		INDICATOR_FWE_BRG := FALSE;
		INDICATOR_FWE_MCR := FALSE;
		INDICATOR_FWE_LC := FALSE;
	(*current status is STANDBY*)
	ELSIF   AUX_EOT_STATUS = 1
	THEN
		(*All the “STAND BY” indicators should keep stable light*)
		INDICATOR_STANDBY_BRG := TRUE;
		INDICATOR_STANDBY_MCR := TRUE;
		INDICATOR_STANDBY_LC := TRUE;
		(*other indicators should keep light off*)
		INDICATOR_ATSEA_BRG := FALSE;
		INDICATOR_ATSEA_MCR := FALSE;
		INDICATOR_ATSEA_LC := FALSE;
		INDICATOR_FWE_BRG := FALSE;
		INDICATOR_FWE_MCR := FALSE;
		INDICATOR_FWE_LC := FALSE;
	(*current status is ATSEA*)
	ELSIF  AUX_EOT_STATUS = 2
	THEN
		(*All the “AT SEA” indicators should keep stable light*)
		INDICATOR_ATSEA_BRG := TRUE;
		INDICATOR_ATSEA_MCR := TRUE;
		INDICATOR_ATSEA_LC := TRUE;
		(*other indicators should keep light off*)
		INDICATOR_STANDBY_BRG := FALSE;
		INDICATOR_STANDBY_MCR := FALSE;
		INDICATOR_STANDBY_LC := FALSE;
		INDICATOR_FWE_BRG := FALSE;
		INDICATOR_FWE_MCR := FALSE;
		INDICATOR_FWE_LC := FALSE;
	(*current status is F.W.E*)
	ELSIF	AUX_EOT_STATUS = 3
	THEN
		(*All the 'FWE” indicators should keep stable light*)
		INDICATOR_FWE_BRG := TRUE;
		INDICATOR_FWE_MCR := TRUE;
		INDICATOR_FWE_LC := TRUE;
		(*other indicators should keep light off*)
		INDICATOR_STANDBY_BRG := FALSE;
		INDICATOR_STANDBY_MCR := FALSE;
		INDICATOR_STANDBY_LC := FALSE;
		INDICATOR_ATSEA_BRG := FALSE;
		INDICATOR_ATSEA_MCR := FALSE;
		INDICATOR_ATSEA_LC := FALSE;
	END_IF
END_IF


CASE AUX_EOT_STATUS OF
	(*none status*)
	0:	H_AT_SEA := FALSE;	(*PROEOT0003*)
		H_STAND_BY := FALSE;	(*PROEOT0004*)
		H_FINSHED_WITH_ENGINE := FALSE;	(*PROEOT0005*)
	(*STAND BY*)
	1:	H_AT_SEA := FALSE;
		H_STAND_BY := TRUE;
		H_FINSHED_WITH_ENGINE := FALSE;
	(*AT SEA*)
	2:	H_AT_SEA := TRUE;
		H_STAND_BY := FALSE;
		H_FINSHED_WITH_ENGINE := FALSE;
	(*FWE*)
	3:	H_AT_SEA := FALSE;
		H_STAND_BY := FALSE;
		H_FINSHED_WITH_ENGINE := TRUE;
END_CASE;
END_FUNCTION_BLOCK

(* POU MISMATCH_ALARM, ST *)
(*4.1.7.1.4*)
FUNCTION_BLOCK MISMATCH_ALARM
VAR_INPUT
END_VAR
VAR_OUTPUT
END_VAR
VAR
	TEMP1: REAL := 0;
	TEMP2: REAL := 0;

	(*mismatch process  flag*)
	MISMATCH_FLAG: BOOL;

	(*mismatch alarm timer, after 1s,slience alarm*)
	ALARM_TIMER: TON;

	(*mismatch alarm occured*)
	MISMATCH_ALARM_FLAG: BOOL;
END_VAR
(*4.1.7.1.4*)
(*自FW*)

TEMP1 := 0;
(*TEMP2 := 0;*)
(*当控制权在BR时,为BR MLV 与 LC MVL 比较,当控制权在MCR_AUTO时，为BR MVL 与 ECR MVL 比较,. 当控制权在LC 时,为LC 与 LC本身比较,不会失步报警*)
(*TEMP1 :=ABS (WORD_TO_REAL( TELEGRAPH_INDICATOR_BR) - WORD_TO_REAL( TELEGRAPH_POSITION_LC));*)


TELEGRAPH_ORDER_THRESHOLD_INPUT := 2 * AD_Scale; (*2mA*)


(*添加当控制权在MCR时,  失步对比选择TELEGRAPH POSITION BR - TELEGRAPG POSITION CR, 并且TELEGRAPH_INDICATOR_BR 与 TELEGRAPH_POSITION_LC ----------begin*)
IF  ECR_AUT_CTRL OR ECR_MAN_CONTROL
THEN
	(*ctrl  in  ECR*)
	(*TEMP1 :=	ABS (WORD_TO_REAL( TELEGRAPH_INDICATOR_BR) - WORD_TO_REAL( TELEGRAPH_POSITION_LC));*)
	TEMP1 :=	ABS (WORD_TO_REAL( TELEGRAPH_POSITION_BR) - WORD_TO_REAL( TELEGRAPH_POSITION_CR));

ELSIF LOCAL_MAN_CTRL THEN
	TEMP1 :=	ABS (WORD_TO_REAL( TELEGRAPH_INDICATOR_BR) - WORD_TO_REAL( TELEGRAPH_POSITION_LC));

END_IF

IF  (ABS(TEMP1) - TELEGRAPH_ORDER_THRESHOLD_INPUT) > 0
	THEN
		MISMATCH_ALARM_FLAG := TRUE;
	ELSE
		MISMATCH_ALARM_FLAG := FALSE;
	END_IF
(*---------------end--------------*)


IF MISMATCH_ALARM_FLAG = TRUE
THEN
	IF  MISMATCH_FLAG = FALSE
	THEN
		IF	BRG_CENR_IN_CONTROL = TRUE
		THEN
			TELEGRAPH_ORDER_BR := TRUE;
		ELSIF	BRG_PORT_IN_CONTROL = TRUE
		THEN
			TELEGRAPH_ORDER_PORT := TRUE;
		ELSIF	BRG_STBD_IN_CONTROL = TRUE
		THEN
			TELEGRAPH_ORDER_STBD := TRUE;
		END_IF

		TELEGRAPH_ORDER_ECR := TRUE;
		TELEGRAPH_ORDER_LC := TRUE;
		TELEGRAPH_COINCIDENCE := FALSE;(*FALSE IS MISMATCH*)

		(*set mismatch  process flag  true*)
		MISMATCH_FLAG := TRUE;
	END_IF

	(*if current ctrl in bridge, then start ALARM timer*)
	IF	BRG_IN_CONTROL_P = TRUE
	THEN
		(*start  alarm timer WHEN ctrl in  bridge*)
		ALARM_TIMER(IN := TRUE, PT := T#60S);
	ELSE
		ALARM_TIMER(IN := FALSE, PT := T#60S);
	END_IF
ELSE
	TELEGRAPH_ORDER_BR := FALSE;
	TELEGRAPH_ORDER_PORT := FALSE;
	TELEGRAPH_ORDER_STBD := FALSE;

	TELEGRAPH_ORDER_ECR := FALSE;
	TELEGRAPH_ORDER_LC := FALSE;


	TELEGRAPH_COINCIDENCE := TRUE;

	(*set mismatch  process flag  FALSE*)
	MISMATCH_FLAG := FALSE;

	(*stop alarm timer*)
	ALARM_TIMER(IN := FALSE);
END_IF


(*Silence telegraph order*)
IF	ESS_BR_ALARM_ACK_P = TRUE
THEN
	TELEGRAPH_ORDER_BR := FALSE;
ELSIF	ESS_ECR_ALARM_ACK_P = TRUE
THEN
	TELEGRAPH_ORDER_ECR := FALSE;
ELSIF	ESS_PORT_ALARM_ACK_P = TRUE
THEN
	TELEGRAPH_ORDER_PORT := FALSE;
ELSIF	ESS_STBD_ALARM_ACK_P = TRUE
THEN
	TELEGRAPH_ORDER_STBD := FALSE;
END_IF

(*after 60s  slicenc mismatch alarm*)
IF  ALARM_TIMER.Q = TRUE
THEN
	TELEGRAPH_ORDER_BR := FALSE;
	TELEGRAPH_ORDER_PORT := FALSE;
	TELEGRAPH_ORDER_STBD := FALSE;

	TELEGRAPH_ORDER_ECR := FALSE;
	TELEGRAPH_ORDER_LC := FALSE;

	ALARM_TIMER(IN := FALSE);
END_IF
END_FUNCTION_BLOCK

(* POU EOT_system_failure_Alarm, ST *)
(*4.1.7.1.5*)
FUNCTION_BLOCK EOT_system_failure_Alarm
VAR_INPUT
END_VAR
VAR_OUTPUT
END_VAR
VAR
END_VAR
(*4.1.7.1.5*)

(*2mA*)
PASSIVE_FAIL_THRESHOLD :=	 2 * AD_Scale; (*2mA*)

(*PASSIVE_FAILURE_BR*)
(*center*)
IF CENT_EOT_MVL > PASSIVE_FAIL_THRESHOLD
THEN
	PASSIVE_FAILURE_BR := FALSE;
ELSE
	PASSIVE_FAILURE_BR := TRUE;
END_IF

IF PORT_WING_EOT_MVL > PASSIVE_FAIL_THRESHOLD
THEN
	PASSIVE_FAILURE_BR_PORT := FALSE;
ELSE
	PASSIVE_FAILURE_BR_PORT := TRUE;
END_IF


IF STBD_WING_EOT_MVL > PASSIVE_FAIL_THRESHOLD
THEN
	PASSIVE_FAILURE_BR_STBD := FALSE;
ELSE
	PASSIVE_FAILURE_BR_STBD := TRUE;
END_IF

(*PASSIVE_FAILURE_ECR*)
IF TELEGRAPH_POSITION_CR > PASSIVE_FAIL_THRESHOLD
THEN
	PASSIVE_FAILURE_ECR := FALSE;
ELSE
	PASSIVE_FAILURE_ECR := TRUE;
END_IF

(*PASSIVE_FAILURE_LC*)
IF TELEGRAPH_POSITION_LC > PASSIVE_FAIL_THRESHOLD
THEN
	PASSIVE_FAILURE_LC := FALSE;
ELSE
	PASSIVE_FAILURE_LC := TRUE;
END_IF

(*TELEGRAPH_SYSTEM_FAIL*)
TELEGRAPH_SYSTEM_FAIL_XS9021A := PASSIVE_FAILURE_BR
											 OR PASSIVE_FAILURE_ECR
											 OR PASSIVE_FAILURE_LC
											 OR PASSIVE_FAILURE_BR_PORT
											 OR PASSIVE_FAILURE_BR_STBD;
END_FUNCTION_BLOCK

(* POU LAMP_TEST, ST *)
FUNCTION_BLOCK LAMP_TEST
VAR_INPUT
END_VAR
VAR_OUTPUT
END_VAR
VAR
END_VAR
(****程序已在其他位置处理好试灯指令,不再用该函数块****)
(*this function block  used to handle the test lamp signal  from  modbus*)
(*-----------------ECR LAMP TEST PB------------------*)
	(*NOT during  transfer MODE*)
IF  MODE_TRANSFER_FLAG = FALSE
THEN
	IF  ECR_LAMP_TEST_PB = TRUE
	THEN
		(*ECR indicator  turn on,buzzer  on*)
		INDICATOR_STANDBY_MCR :=  TRUE;
		INDICATOR_ATSEA_MCR := TRUE;
		INDICATOR_FWE_MCR := TRUE;

		BUZZER_MCR := TRUE;
	ELSE
		(*buzzer  silence*)
		BUZZER_MCR := FALSE;
		(*current status is none*)
		IF AUX_EOT_STATUS = 0
		THEN
			INDICATOR_STANDBY_MCR :=  FALSE;
			INDICATOR_ATSEA_MCR := FALSE;
			INDICATOR_FWE_MCR := FALSE;
		(*current status is STABDBY*)
		ELSIF  AUX_EOT_STATUS = 1
		THEN
			INDICATOR_STANDBY_MCR :=  TRUE;
			INDICATOR_ATSEA_MCR := FALSE;
			INDICATOR_FWE_MCR := FALSE;
		(*current status is ATSEA*)
		ELSIF  AUX_EOT_STATUS = 2
		THEN
			INDICATOR_STANDBY_MCR :=  FALSE;
			INDICATOR_ATSEA_MCR := TRUE;
			INDICATOR_FWE_MCR := FALSE;
		(*current status is FWE*)
		ELSIF  AUX_EOT_STATUS = 3
		THEN
			INDICATOR_STANDBY_MCR :=  FALSE;
			INDICATOR_ATSEA_MCR := FALSE;
			INDICATOR_FWE_MCR := TRUE;
		END_IF
	END_IF
END_IF

(*-----------------BR CENTER LAMP TEST PB------------------*)
(*NOT during  transfer AND bridge control  positon change  process*)
IF	MODE_TRANSFER_FLAG = FALSE
	AND  CONTROL_TRANS_PROCESS_FLAG = FALSE
THEN
	IF	BR_LAMP_TEST_PB = TRUE
	THEN
		(*bridge  center  indicator  all off,buzzer  on*)
		INDICATOR_STANDBY_BRG := TRUE;
		INDICATOR_ATSEA_BRG := TRUE;
		INDICATOR_FWE_BRG := TRUE;

		BRIDGE_PORT_EOT_IN_CONTROL_LAMP := TRUE;
		BRIDGE_STBD_EOT_IN_CONTROL_LAMP := TRUE;

		BUZZER_BRG := TRUE;
		BRIDGE_BUZZER := TRUE;
	ELSE
		(*buzzer  silence*)
		BUZZER_BRG := FALSE;
		BRIDGE_BUZZER := FALSE;

		(*current status is none*)
		IF AUX_EOT_STATUS = 0
		THEN
			INDICATOR_STANDBY_BRG :=  FALSE;
			INDICATOR_ATSEA_BRG := FALSE;
			INDICATOR_FWE_BRG := FALSE;
		(*current status is STABDBY*)
		ELSIF  AUX_EOT_STATUS = 1
		THEN
			INDICATOR_STANDBY_BRG :=  TRUE;
			INDICATOR_ATSEA_BRG := FALSE;
			INDICATOR_FWE_BRG := FALSE;
		(*current status is ATSEA*)
		ELSIF  AUX_EOT_STATUS = 2
		THEN
			INDICATOR_STANDBY_BRG :=  FALSE;
			INDICATOR_ATSEA_BRG := TRUE;
			INDICATOR_FWE_BRG := FALSE;
		(*current status is FWE*)
		ELSIF  AUX_EOT_STATUS = 3
		THEN
			INDICATOR_STANDBY_BRG :=  FALSE;
			INDICATOR_ATSEA_BRG := FALSE;
			INDICATOR_FWE_BRG := TRUE;
		END_IF
	END_IF
END_IF


(*-----------------BR PORT LAMP TEST PB------------------*)
 (*NOT during bridge control  positon change  process*)
IF  CONTROL_TRANS_PROCESS_FLAG = FALSE
THEN
	IF	PORT_LAMP_TEST_PB = TRUE
	THEN
		PORT_EOT_IN_CONTROL_LAMP := TRUE;
		PORT_BUZZER := TRUE;
	ELSE
		PORT_BUZZER := FALSE;
	END_IF
END_IF

(*-----------------STBD PORT LAMP TEST PB------------------*)
(*NOT during bridge control  positon change  process*)
IF  CONTROL_TRANS_PROCESS_FLAG = FALSE
THEN
	IF	STBD_LAMP_TEST_PB = TRUE
	THEN
		STBD_EOT_IN_CONTROL_LAMP := TRUE;
		STBD_BUZZER := TRUE;
	ELSE
		STBD_BUZZER := FALSE;
	END_IF
END_IF
END_FUNCTION_BLOCK

(* POU AMPERE_STAGE_TO_HMI, ST *)
FUNCTION_BLOCK AMPERE_STAGE_TO_HMI
VAR_INPUT
END_VAR
VAR_OUTPUT
END_VAR
VAR
	TON_Init: TON;

	(*all stage limit bound.  4 -- 20ma*)
	Emergency_AS_LOW: REAL;
	Emergency_AS_HIGH: REAL;

	Full_AS_LOW: REAL;
	Full_AS_HIGH: REAL;

	HALF_AS_LOW: REAL;
	HALF_AS_HIGH: REAL;

	SLOW_AS_LOW: REAL;
	SLOW_AS_HIGH: REAL;

	DS_S_AS_LOW: REAL;
	DS_S_AS_HIGH: REAL;

	STOP_LOW: REAL;
	STOP_HIGH: REAL;

	DEAD_S_AH_LOW: REAL;
	DEAD_S_AH_HIGH: REAL;

	SLOW_AH_LOW: REAL;
	SLOW_AH_HIGH: REAL;

	HALF_AH_LOW: REAL;
	HALF_AH_HIGH: REAL;

	Full_AH_LOW: REAL;
	Full_AH_HIGH: REAL;

	Full_SEA_AH_LOW: REAL;
	Full_SEA_AH_HIGH: REAL;

	(*valid stage  counts, get sample 10 times *)
	stage_change_cnts: BYTE;

	(*11 stage valid  counts array,  array[0] is  Emergency AS,  array[10]  is  Full SEA  AH*)
	arStageValidCnt:  ARRAY[0..10] OF BYTE;

	i: BYTE;

END_VAR
(*INIT  in 0.5S*)

TON_Init(IN := TRUE, PT := t#0.5s);

(*INIT  IN  0.5S*)
IF	TON_Init.Q = FALSE
THEN
	(*set  stage  limit   bound*)
	(*all stage limit bound.  4 -- 20ma*)
	Emergency_AS_LOW := 4 * AD_Scale;
	Emergency_AS_HIGH :=  4.5 * AD_Scale;

	Full_AS_LOW := 4.5 * AD_Scale;
	Full_AS_HIGH := 5.5 * AD_Scale;

	HALF_AS_LOW := 5.5 * AD_Scale;
	HALF_AS_HIGH := 7 * AD_Scale;

	SLOW_AS_LOW := 7 * AD_Scale;
	SLOW_AS_HIGH := 9 * AD_Scale;

	DS_S_AS_LOW := 9 * AD_Scale;
	DS_S_AS_HIGH := 11 * AD_Scale;

	STOP_LOW := 11 * AD_Scale;
	STOP_HIGH := 13 * AD_Scale;

	DEAD_S_AH_LOW := 13 * AD_Scale;
	DEAD_S_AH_HIGH := 15 * AD_Scale;

	SLOW_AH_LOW := 15 * AD_Scale;
	SLOW_AH_HIGH := 17 * AD_Scale;

	HALF_AH_LOW := 17 * AD_Scale;
	HALF_AH_HIGH := 18.5 * AD_Scale;

	Full_AH_LOW  := 18.5 * AD_Scale;
	Full_AH_HIGH := 19.5 * AD_Scale;

	Full_SEA_AH_LOW := 19.5 * AD_Scale;
	Full_SEA_AH_HIGH := 20.5 * AD_Scale;

	RETURN ;
END_IF


(***程序每次周期(20ms)运行采集当前输入电流值并判断属于哪个档位区间,在10个周期内(200ms)采集10次,若10次电流值均位于同一档位区间,则认为该档位有效,主要用于消除抖动***)
(*********judge  current  stage,  every cycle  sampling the  TELEGRAPH_INDICATOR_BR, and  store it  in  the corresponding  ARRAY position***********)
(*Emergency AS*)
IF	TELEGRAPH_POSITION_BR >=  Emergency_AS_LOW
	AND  TELEGRAPH_POSITION_BR <  Emergency_AS_HIGH
THEN
	arStageValidCnt[0] := arStageValidCnt[0] + 1;
(*FULL  AS*)
ELSIF	TELEGRAPH_POSITION_BR >= Full_AS_LOW
	AND  TELEGRAPH_POSITION_BR < Full_AS_HIGH
THEN
	arStageValidCnt[1] := arStageValidCnt[1] + 1;
(*HALF  AS*)
ELSIF	TELEGRAPH_POSITION_BR >= HALF_AS_LOW
	AND  TELEGRAPH_POSITION_BR < HALF_AS_HIGH
THEN
	arStageValidCnt[2] := arStageValidCnt[2] + 1;
(*SLOW_AS*)
ELSIF	TELEGRAPH_POSITION_BR >= SLOW_AS_LOW
	AND  TELEGRAPH_POSITION_BR < SLOW_AS_HIGH
THEN
	arStageValidCnt[3] := arStageValidCnt[3] + 1;
(*DS_S_AS*)
ELSIF	TELEGRAPH_POSITION_BR >= DS_S_AS_LOW
	AND  TELEGRAPH_POSITION_BR < DS_S_AS_HIGH
THEN
	arStageValidCnt[4] := arStageValidCnt[4] + 1;
(*STOP*)
ELSIF	TELEGRAPH_POSITION_BR >= STOP_LOW
	AND  TELEGRAPH_POSITION_BR < STOP_HIGH
THEN
	arStageValidCnt[5] := arStageValidCnt[5] + 1;
(*DEAD_S_AH*)
ELSIF	TELEGRAPH_POSITION_BR >= DEAD_S_AH_LOW
	AND  TELEGRAPH_POSITION_BR < DEAD_S_AH_HIGH
THEN
	arStageValidCnt[6] := arStageValidCnt[6] + 1;
(*SLOW_AH*)
ELSIF	TELEGRAPH_POSITION_BR >= SLOW_AH_LOW
	AND  TELEGRAPH_POSITION_BR < SLOW_AH_HIGH
THEN
	arStageValidCnt[7] := arStageValidCnt[7] + 1;
(*HALF_AH*)
ELSIF	TELEGRAPH_POSITION_BR >= HALF_AH_LOW
	AND  TELEGRAPH_POSITION_BR < HALF_AH_HIGH
THEN
	arStageValidCnt[8] := arStageValidCnt[8] + 1;
(*Full_AH*)
ELSIF	TELEGRAPH_POSITION_BR >= Full_AH_LOW
	AND  TELEGRAPH_POSITION_BR < Full_AH_HIGH
THEN
	arStageValidCnt[9] := arStageValidCnt[9] + 1;
(*Full_SEA_AH*)
ELSIF	TELEGRAPH_POSITION_BR >= Full_SEA_AH_LOW
	AND  TELEGRAPH_POSITION_BR <= Full_SEA_AH_HIGH
THEN
	arStageValidCnt[10] := arStageValidCnt[10] + 1;
END_IF

(*sampling  times count*)
stage_change_cnts := stage_change_cnts + 1;

(*after  sampling  10  times,  judge  the  current  stage is  valid or  not*)
IF	stage_change_cnts = 10
THEN
	AMPERE_STAGE_TO_HMI := 0;
	FOR  i := 0 TO 10 BY 1 DO
		IF	arStageValidCnt[i] = 10
		THEN
			AMPERE_STAGE_TO_HMI := SHL(WORD#1, i);
		END_IF

		(*clear stage valid  counts array*)
		arStageValidCnt[i] := 0;
	END_FOR

	(*restart  count  sampling  times*)
	stage_change_cnts := 0;
END_IF

Telegraph_Indicator_Full_SEA_AH :=  WORD_TO_BOOL(SHR(AMPERE_STAGE_TO_HMI AND 16#400, 10));
Telegraph_Indicator_FULL_AH :=  WORD_TO_BOOL(SHR(AMPERE_STAGE_TO_HMI AND 16#200, 9));
Telegraph_Indicator_HALF_AH :=  WORD_TO_BOOL(SHR(AMPERE_STAGE_TO_HMI AND 16#100, 8));
Telegraph_Indicator_SLOW_AH :=  WORD_TO_BOOL(SHR(AMPERE_STAGE_TO_HMI AND 16#80, 7));
Telegraph_Indicator_DEAD_S_AH :=  WORD_TO_BOOL(SHR(AMPERE_STAGE_TO_HMI AND 16#40, 6));
Telegraph_Indicator_STOP :=  WORD_TO_BOOL(SHR(AMPERE_STAGE_TO_HMI AND 16#20, 5));
Telegraph_Indicator_DEAD_S_AS :=  WORD_TO_BOOL(SHR(AMPERE_STAGE_TO_HMI AND 16#10, 4));
Telegraph_Indicator_SLOW_AS :=  WORD_TO_BOOL(SHR(AMPERE_STAGE_TO_HMI AND 16#8, 3));
Telegraph_Indicator_HALF_AS :=  WORD_TO_BOOL(SHR(AMPERE_STAGE_TO_HMI AND 16#4, 2));
Telegraph_Indicator_FULL_AS :=  WORD_TO_BOOL(SHR(AMPERE_STAGE_TO_HMI AND 16#2, 1));
Telegraph_Indicator_Emergency_AS :=  WORD_TO_BOOL(SHR(AMPERE_STAGE_TO_HMI AND 16#1, 0));
END_FUNCTION_BLOCK

(* POU MVL_COMMD_TO_AO, ST *)
FUNCTION_BLOCK MVL_COMMD_TO_AO
VAR_INPUT
END_VAR
VAR_OUTPUT
END_VAR
VAR
	Real_Current: REAL;
END_VAR
(***********TO  RCS**********)
(**** BR****)
(*将输入数字量转化为电流值, 若AI模块范围为4~20mA,则电流值应+4, 若AI模块范围为0~20mA,则电流值不加4*)
Real_Current := WORD_TO_REAL( TELEGRAPH_POSITION_BR) / AD_Scale;

(*将电流值转化为输出数字量, 若AO模块范围为4~20mA,则电流值应-4, 若AO模块范围为0~20mA,则电流值不-4*)
BR_MVL_COMMD_TO_RCS_P :=  REAL_TO_WORD((Real_Current -4) * DA_Scale);


(**** ECR****)
(*将输入数字量转化为电流值, 若AI模块范围为4~20mA,则电流值应+4, 若AI模块范围为0~20mA,则电流值不加4*)
Real_Current := WORD_TO_REAL (TELEGRAPH_POSITION_CR) / AD_Scale;

(*将电流值转化为输出数字量, 若AO模块范围为4~20mA,则电流值应-4, 若AO模块范围为0~20mA,则电流值不-4*)
ECR_MVL_COMMD_TO_RCS_P :=  REAL_TO_WORD((Real_Current-4) * DA_Scale);


(**********INDICATOR  TO AO*****************)
(****BR  INDICATOR****)
(*将输入数字量转化为电流值, 若AI模块范围为4~20mA,则电流值应+4, 若AI模块范围为0~20mA,则电流值不加4*)
Real_Current := WORD_TO_REAL( TELEGRAPH_INDICATOR_BR) / AD_Scale;

(*将电流值转化为输出数字量, 若AO模块范围为4~20mA,则电流值应-4, 若AO模块范围为0~20mA,则电流值不-4*)
BR_Indicator_Position_Pointer_P :=  REAL_TO_WORD((Real_Current -4) * DA_Scale);

(****ECR  INDICATOR****)
(*将输入数字量转化为电流值, 若AI模块范围为4~20mA,则电流值应+4, 若AI模块范围为0~20mA,则电流值不加4*)
Real_Current := WORD_TO_REAL( TELEGRAPH_INDICATOR_ECR) / AD_Scale;

(*将电流值转化为输出数字量, 若AO模块范围为4~20mA,则电流值应-4, 若AO模块范围为0~20mA,则电流值不-4*)
ECR_Indicator_Position_Pointer_P :=  REAL_TO_WORD((Real_Current -4) * DA_Scale);

(****LC  INDICATOR****)
(*将输入数字量转化为电流值, 若AI模块范围为4~20mA,则电流值应+4, 若AI模块范围为0~20mA,则电流值不加4*)
Real_Current := WORD_TO_REAL( TELEGRAPH_INDICATOR_LC) / AD_Scale;

(*将电流值转化为输出数字量, 若AO模块范围为4~20mA,则电流值应-4, 若AO模块范围为0~20mA,则电流值不-4*)
LOCAL_Indicator_Position_Pointer_P :=  REAL_TO_WORD((Real_Current -4) * DA_Scale);

(***BR	PORT INDICATOR****)
(*将输入数字量转化为电流值, 若AI模块范围为4~20mA,则电流值应+4, 若AI模块范围为0~20mA,则电流值不加4*)
Real_Current := WORD_TO_REAL( TELEGRAPH_INDICATOR_BR_PORT) / AD_Scale;

(*将电流值转化为输出数字量, 若AO模块范围为4~20mA,则电流值应-4, 若AO模块范围为0~20mA,则电流值不-4*)
BR_PORT_Indicator_Position_Pointer_P :=  REAL_TO_WORD((Real_Current -4) * DA_Scale);

(***BR	STBD  INDICATOR****)
(*将输入数字量转化为电流值, 若AI模块范围为4~20mA,则电流值应+4, 若AI模块范围为0~20mA,则电流值不加4*)
Real_Current := WORD_TO_REAL( TELEGRAPH_INDICATOR_BR_STBD) / AD_Scale;

(*将电流值转化为输出数字量, 若AO模块范围为4~20mA,则电流值应-4, 若AO模块范围为0~20mA,则电流值不-4*)
BR_STBD_Indicator_Position_Pointer_P :=  REAL_TO_WORD((Real_Current -4) * DA_Scale);


(*TEST  吴凡让加的*)
(*将输入数字量转化为电流值, 若AI模块范围为4~20mA,则电流值应+4, 若AI模块范围为0~20mA,则电流值不加4*)
Real_Current := WORD_TO_REAL( TELEGRAPH_POSITION_LC) / AD_Scale;

(*将电流值转化为输出数字量, 若AO模块范围为4~20mA,则电流值应-4, 若AO模块范围为0~20mA,则电流值不-4*)
TEST_LOCAL_Telegraph_Position_Pointer_P :=  REAL_TO_WORD((Real_Current -4) * DA_Scale);
END_FUNCTION_BLOCK

(* POU MVL_TO_RCS_TEST_MBS, ST *)
FUNCTION_BLOCK MVL_TO_RCS_TEST_MBS
VAR_INPUT
END_VAR
VAR_OUTPUT
END_VAR
VAR
END_VAR
BR_MVL_TO_RCS_MBS_P	:=  TELEGRAPH_POSITION_BR;
ECR_MVL_TO_RCS_MBS_P :=  TELEGRAPH_POSITION_CR;


BR_MVL_TO_RCS_MBS_P1	:=	BR_MVL_TO_RCS_MBS_P;
ECR_MVL_TO_RCS_MBS_P1 :=	ECR_MVL_TO_RCS_MBS_P;
END_FUNCTION_BLOCK
